Fanuc KAREL source: kt00891.KL

-- PROVISIONAL review KL for V770-1; original PC SHA256 679383c3d9aef75da5de894d82fbfb7c9b83e26ba561f96638d8116e853d6e8c
-- Incomplete behavior may be omitted. Consult companion uncertainty JSON. Do not deploy.
PROGRAM KT00891
%NOLOCKGROUP
-- UNRESOLVED_DECL P1 type=000199
-- UNRESOLVED_DECL P2 type=000199
-- UNRESOLVED_DECL OUT type=000101
BEGIN
  -- UNRESOLVED_PC offsets 5-35; opcodes 27,27,49,7E,AD,76,7E,4A
  -- UNRESOLVED_PC offsets 40-44; opcodes 7F
END KT00891
